Universal Robots PolyScope program: test protective stop.urp

Program test protective stop (installation=default directory=/programs createdIn=5.14.5 lastSavedIn=5.14.5 robotSerialNumber=20236801216)
Calibrated DH parameters: a=[-0.000021, -0.748897, -0.28186, -0.00004, -0.000055, 0]; d=[0.236225, -424.082933, -1564.66872, 1988.95162, 0.159094, 0.153873]; alpha=[1.570844, 0.001002, 0.000337, 1.571488, -1.569996, 0]; deltaTheta=[0, -0.516316, 5.626292, 1.173211, 0.000001, 0]
InitVariablesNode
BeforeStart
  Set NoAction tcp=pretend_welder
Robot Program (runOnlyOnce=false)
  MoveJ speed 60 deg/s, acceleration 80 deg/s^2 (useActiveTCP=true) feature=Base
    Waypoint Waypoint_1: TCP in base x=82.42 y=948.23 z=435.005 mm, rx=0.9103 ry=2.9915 rz=0.081 rad; joints [-123.873, -69.54, 91.006, 63.378, -0.135, -87.909] deg; TCP offset x=4.51 y=-328 z=106.39 mm, rx=1.2092 ry=-1.2092 rz=1.2092 rad
  Wait Sleep waitTime=1
  MoveJ speed 60 deg/s, acceleration 80 deg/s^2 (useActiveTCP=true) feature=Base
    Waypoint Waypoint_2: TCP in base x=-203.248 y=523.643 z=235.567 mm, rx=-0.8211 ry=-2.695 rz=0.8924 rad; joints [-123.873, -69.539, 130.755, 63.379, -0.136, -87.91] deg
SuppressedNode
  Thread Thread_1 (runOnlyOnce=false)
    If is_protective_stop()
      pts := True
    Else 
      pts := False
